(* Logix 5000 project; controller PLC_Safety vendor 1 type 14 code 148 rev 37.11; software revision 37.00; part 2 of 3 *)
(* tags used below, declared in another part *)
   Contador_num_pza : COUNTER;
   Contador_pza_aprove : COUNTER;
   Contador_pza_rechazada : COUNTER;
   Counter_Parts : COUNTER;   // Trazabilidad
   Done_cicle : BOOL;
   FANUC_R1 : BOOL;
   FANUC_R2 : BOOL;
   FANUC_R3 : BOOL;
   FANUC_R4 : BOOL;
   Fanuc_Strobe : BOOL;
   HMI_Cognex_medio : DINT;   // HMI
   HMI_Fanucbrazo : DINT;   // HMI
   HMI_Fanucdelta : DINT;   // HMI
   HMI_Fcognexmedio : BOOL;   // HMI
   HMI_Ffanucbrazo : BOOL;   // HMI
   HMI_Ffanucdelta : BOOL;   // HMI
   HMI_Fplc1 : BOOL;   // HMI
   HMI_Fplc2 : BOOL;   // HMI
   HMI_Fplcseguridad : BOOL;   // HMI
   HMI_kinetix1 : BOOL;   // HMI
   HMI_kinetix2 : BOOL;
   HMI_Kinetix_1 : DINT;   // HMI
   HMI_Kinetix_2 : DINT;
   HMI_PLC1 : DINT;   // HMI
   HMI_PLC2 : DINT;   // HMI
   HMI_PLC_Seguridad : DINT;   // HMI
   HMI_PointIO1 : BOOL;   // HMI
   HMI_PointIO2 : BOOL;
   HMI_PointIO3 : BOOL;
   HMI_PointIO4 : BOOL;
   HMI_PointIO6 : BOOL;
   HMI_PointIO_1 : DINT;   // HMI
   HMI_PointIO_2 : DINT;
   HMI_PointIO_3 : DINT;
   HMI_PointIO_4 : DINT;
   HMI_PointIO_6 : DINT;
   HMI_R_cognex1 : BOOL;
   HMI_R_cognex2 : BOOL;
   HMI_R_PF1 : BOOL;
   HMI_R_PF2 : BOOL;
   HMI_S_cognex1 : BOOL;
   HMI_S_cognex2 : BOOL;
   HMI_S_PF1 : BOOL;
   HMI_S_PF2 : BOOL;
   HMI_Switch1 : BOOL;
   HMI_Switch2 : BOOL;
   HMI_Switch3 : BOOL;
   HMI_Switch4 : BOOL;
   HMI_Switch5 : BOOL;
   OSF_Fault_Reset_Fanuc : BOOL;
   Part : REAL;
   Piece_Approved : BOOL;
   Piece_Base : BOOL;
   Piece_Coil : BOOL;
   Piece_Rejected : BOOL;
   Piece_Upper : BOOL;
   S2_Height_1 : BOOL;
   S2_Height_2 : BOOL;
   S2_Height_3 : BOOL;
   S2_Height_4 : BOOL;
   S2_Height_5 : BOOL;
   S2_Height_6 : BOOL;
   S2_Height_Conveyor_1 : BOOL;
   S2_Height_Conveyor_2 : BOOL;
   S2_MAM_Height_1 : MOTION_INSTRUCTION;
   S2_MAM_Height_2 : MOTION_INSTRUCTION;
   S2_MAM_Height_3 : MOTION_INSTRUCTION;
   S2_MAM_Height_4 : MOTION_INSTRUCTION;
   S2_MAM_Height_5 : MOTION_INSTRUCTION;
   S2_MAM_Height_6 : MOTION_INSTRUCTION;
   S2_MAM_Height_Conveyor_1 : MOTION_INSTRUCTION;
   S2_MAM_Height_Conveyor_2 : MOTION_INSTRUCTION;
   S2_MSO_Storage : MOTION_INSTRUCTION;
   S2_Sensor_Height_1 : BOOL;
   S2_Sensor_Height_2 : BOOL;
   S2_Sensor_Height_3 : BOOL;
   S2_Sensor_Height_4 : BOOL;
   S2_Sensor_Height_5 : BOOL;
   S2_Sensor_Height_6 : BOOL;
   S2_Sensor_Height_Conveyor_1 : BOOL;
   S2_Sensor_Height_Conveyor_2 : BOOL;
   S2_Storage_On : BOOL;
   Sensor_FANUC_R1 : BOOL;
   Sensor_FANUC_R2 : BOOL;
   Sensor_FANUC_R3 : BOOL;
   Sensor_FANUC_R4 : BOOL;
   Start_Button_1_Secuencia : BOOL;
   Start_Button_2_Secuencia : BOOL;
   Start_Button_3_Secuencia : BOOL;
   Trigger_Cognex_3 : BOOL;
   Axis_2 : AXIS_CIP_DRIVE;   // Storage 2
   Data_From_PLC2 : DINT[20];
   Data_To_PLC1 : DINT[20];
   Data_To_PLC2 : DINT[20];
   E_Stop_1_NC : ALIAS FOR Point_IO_Gabinete_1:6:I.Pt01Data;   // E Stop 1 Normally Close
   E_Stop_1_NO : ALIAS FOR Point_IO_Gabinete_1:6:I.Pt00Data;   // E Stop 1 Normally Open
   E_Stop_2_NC : ALIAS FOR Point_IO_Gabinete_2:6:I.Pt01Data;   // E Stop 2 Normally Close
   E_Stop_2_NO : ALIAS FOR Point_IO_Gabinete_2:6:I.Pt00Data;   // E Stop 2 Normally Open
   E_Stop_3_NC : ALIAS FOR Point_IO_Gabinete_6:4:I.Pt02Data;   // E Stop 3 Normally Close
   E_Stop_3_NO : ALIAS FOR Point_IO_Gabinete_6:4:I.Pt03Data;   // E Stop 3 Normally Open
   E_Stop_Conveyor_1_NC : ALIAS FOR Point_IO_Gabinete_3:11:I.Pt00Data;   // E Stop Conveyor 1 Normally Close
   E_Stop_Conveyor_1_NO : ALIAS FOR Point_IO_Gabinete_3:11:I.Pt01Data;   // E Stop Conveyor 1 Normally Open
   E_Stop_Conveyor_2_NC : ALIAS FOR Point_IO_Gabinete_4:11:I.Pt00Data;   // E Stop Conveyor 2 Normally Close
   E_Stop_Conveyor_2_NO : ALIAS FOR Point_IO_Gabinete_4:11:I.Pt01Data;   // E Stop Conveyor 2 Normally Open
   E_Stop_OK : BOOL;
   Reset_General : BOOL;
   Safety_OK : BOOL;
(* MainProgram, continued *)

ROUTINE R05_Storage_2   (* ladder *)
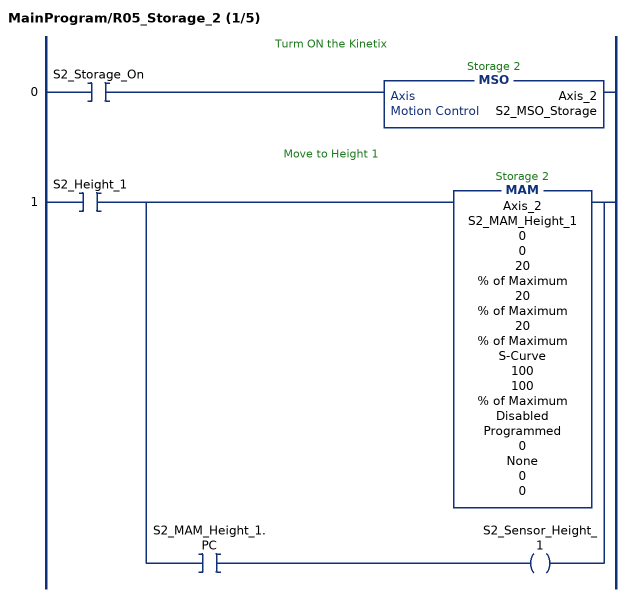
   // Turm ON the Kinetix
   0: XIC(S2_Storage_On)MSO(Axis_2,S2_MSO_Storage);
   // Move to Height 1
   1: XIC(S2_Height_1)[MAM(Axis_2,S2_MAM_Height_1,0,0,20,% of Maximum,20,% of Maximum,20,% of Maximum,S-Curve,100,100,% of Maximum,Disabled,Programmed,0,None,0,0) ,XIC(S2_MAM_Height_1.PC) OTE(S2_Sensor_Height_1) ];
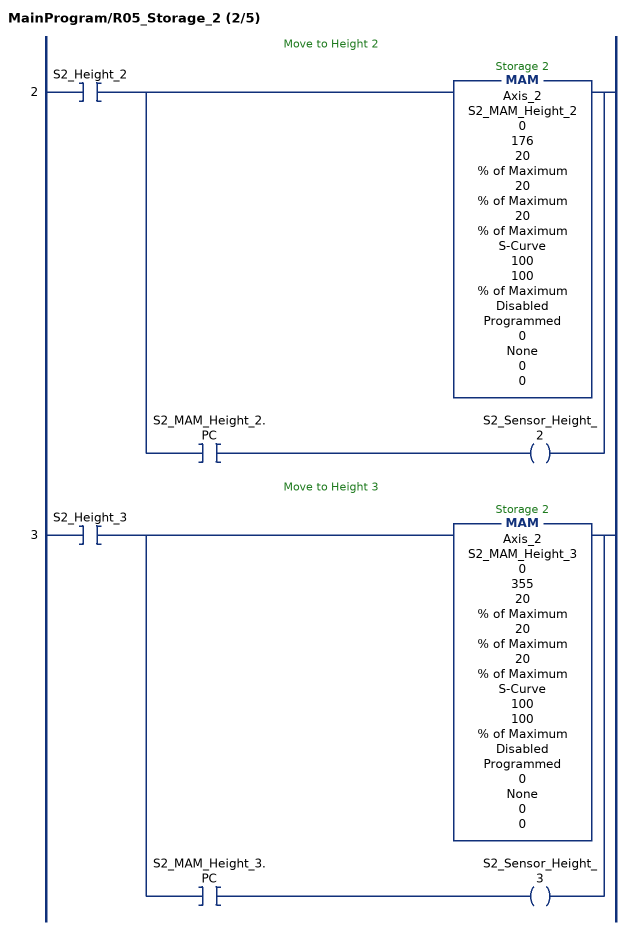
   // Move to Height 2
   2: XIC(S2_Height_2)[MAM(Axis_2,S2_MAM_Height_2,0,176,20,% of Maximum,20,% of Maximum,20,% of Maximum,S-Curve,100,100,% of Maximum,Disabled,Programmed,0,None,0,0) ,XIC(S2_MAM_Height_2.PC) OTE(S2_Sensor_Height_2) ];
   // Move to Height 3
   3: XIC(S2_Height_3)[MAM(Axis_2,S2_MAM_Height_3,0,355,20,% of Maximum,20,% of Maximum,20,% of Maximum,S-Curve,100,100,% of Maximum,Disabled,Programmed,0,None,0,0) ,XIC(S2_MAM_Height_3.PC) OTE(S2_Sensor_Height_3) ];
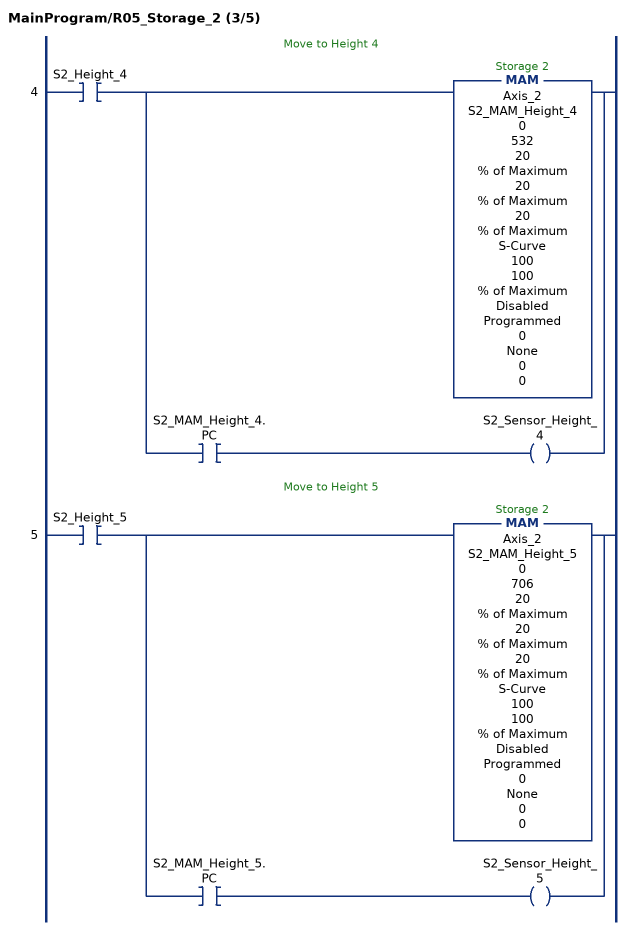
   // Move to Height 4
   4: XIC(S2_Height_4)[MAM(Axis_2,S2_MAM_Height_4,0,532,20,% of Maximum,20,% of Maximum,20,% of Maximum,S-Curve,100,100,% of Maximum,Disabled,Programmed,0,None,0,0) ,XIC(S2_MAM_Height_4.PC) OTE(S2_Sensor_Height_4) ];
   // Move to Height 5
   5: XIC(S2_Height_5)[MAM(Axis_2,S2_MAM_Height_5,0,706,20,% of Maximum,20,% of Maximum,20,% of Maximum,S-Curve,100,100,% of Maximum,Disabled,Programmed,0,None,0,0) ,XIC(S2_MAM_Height_5.PC) OTE(S2_Sensor_Height_5) ];
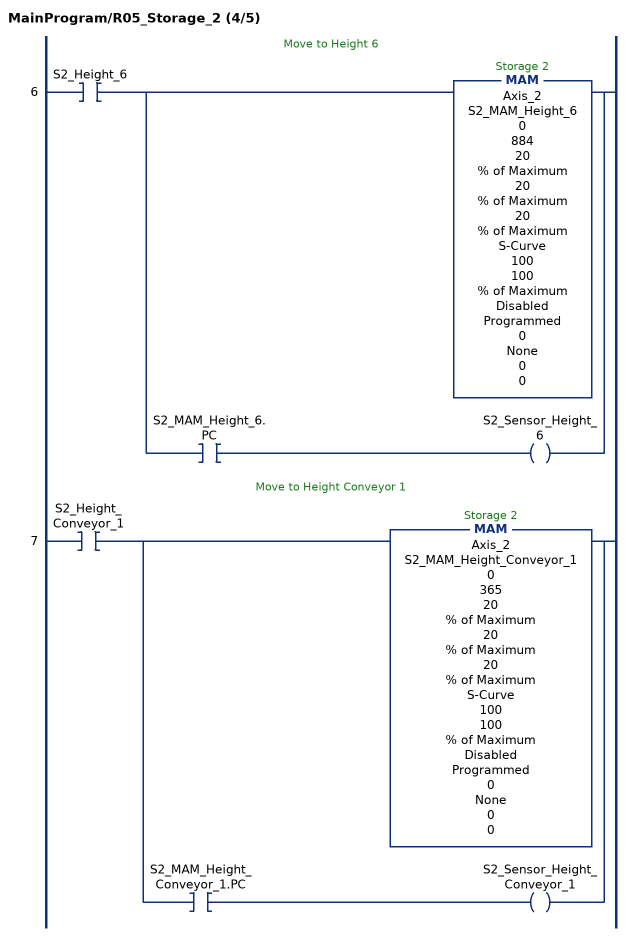
   // Move to Height 6
   6: XIC(S2_Height_6)[MAM(Axis_2,S2_MAM_Height_6,0,884,20,% of Maximum,20,% of Maximum,20,% of Maximum,S-Curve,100,100,% of Maximum,Disabled,Programmed,0,None,0,0) ,XIC(S2_MAM_Height_6.PC) OTE(S2_Sensor_Height_6) ];
   // Move to Height Conveyor 1
   7: XIC(S2_Height_Conveyor_1)[MAM(Axis_2,S2_MAM_Height_Conveyor_1,0,365,20,% of Maximum,20,% of Maximum,20,% of Maximum,S-Curve,100,100,% of Maximum,Disabled,Programmed,0,None,0,0) ,XIC(S2_MAM_Height_Conveyor_1.PC) OTE(S2_Sensor_Height_Conveyor_1) ];
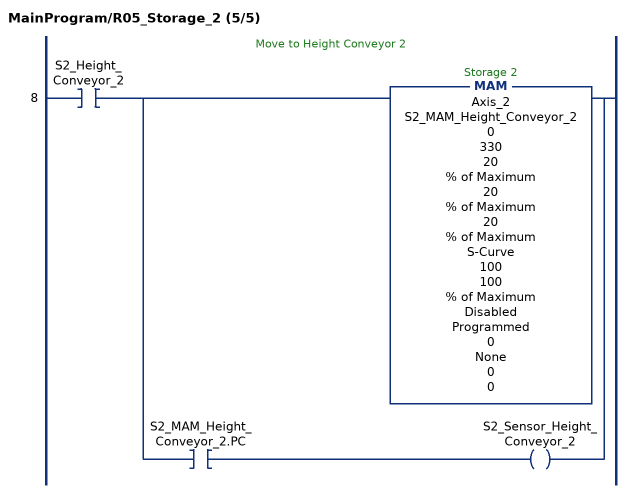
   // Move to Height Conveyor 2
   8: XIC(S2_Height_Conveyor_2)[MAM(Axis_2,S2_MAM_Height_Conveyor_2,0,330,20,% of Maximum,20,% of Maximum,20,% of Maximum,S-Curve,100,100,% of Maximum,Disabled,Programmed,0,None,0,0) ,XIC(S2_MAM_Height_Conveyor_2.PC) OTE(S2_Sensor_Height_Conveyor_2) ];
END_ROUTINE

ROUTINE R06_Fanuc   (* ladder *)
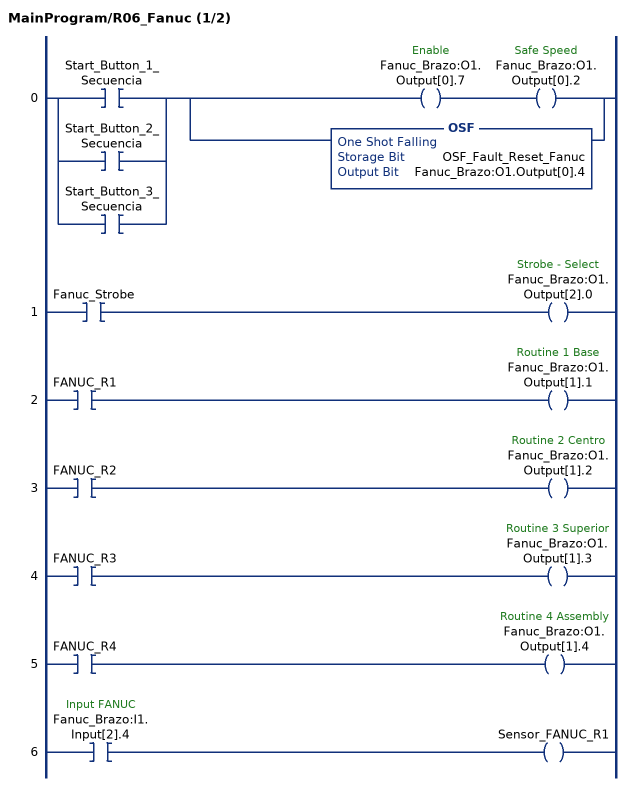
   0: [XIC(Start_Button_1_Secuencia) ,XIC(Start_Button_2_Secuencia) ,XIC(Start_Button_3_Secuencia) ][OTE(Fanuc_Brazo:O1.Output[0].7) OTE(Fanuc_Brazo:O1.Output[0].2) ,OSF(OSF_Fault_Reset_Fanuc,Fanuc_Brazo:O1.Output[0].4) ];
   1: XIC(Fanuc_Strobe)OTE(Fanuc_Brazo:O1.Output[2].0);
   2: XIC(FANUC_R1)OTE(Fanuc_Brazo:O1.Output[1].1);
   3: XIC(FANUC_R2)OTE(Fanuc_Brazo:O1.Output[1].2);
   4: XIC(FANUC_R3)OTE(Fanuc_Brazo:O1.Output[1].3);
   5: XIC(FANUC_R4)OTE(Fanuc_Brazo:O1.Output[1].4);
   6: XIC(Fanuc_Brazo:I1.Input[2].4)OTE(Sensor_FANUC_R1);
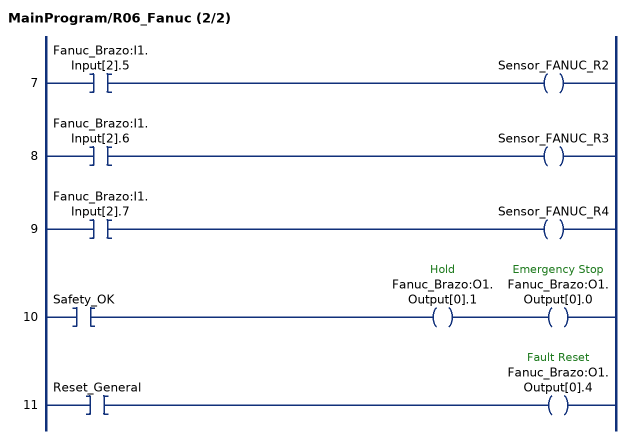
   7: XIC(Fanuc_Brazo:I1.Input[2].5)OTE(Sensor_FANUC_R2);
   8: XIC(Fanuc_Brazo:I1.Input[2].6)OTE(Sensor_FANUC_R3);
   9: XIC(Fanuc_Brazo:I1.Input[2].7)OTE(Sensor_FANUC_R4);
   10: XIC(Safety_OK)OTE(Fanuc_Brazo:O1.Output[0].1)OTE(Fanuc_Brazo:O1.Output[0].0);
   11: XIC(Reset_General)OTE(Fanuc_Brazo:O1.Output[0].4);
END_ROUTINE

ROUTINE R07_Cognex_3   (* ladder *)
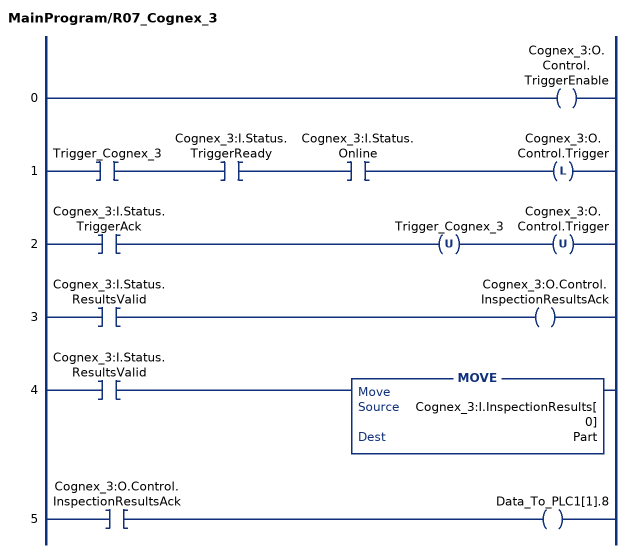
   0: OTE(Cognex_3:O.Control.TriggerEnable);
   1: XIC(Trigger_Cognex_3)XIC(Cognex_3:I.Status.TriggerReady)XIC(Cognex_3:I.Status.Online)OTL(Cognex_3:O.Control.Trigger);
   2: XIC(Cognex_3:I.Status.TriggerAck)OTU(Trigger_Cognex_3)OTU(Cognex_3:O.Control.Trigger);
   3: XIC(Cognex_3:I.Status.ResultsValid)OTE(Cognex_3:O.Control.InspectionResultsAck);
   4: XIC(Cognex_3:I.Status.ResultsValid)MOVE(Cognex_3:I.InspectionResults[0],Part);
   5: XIC(Cognex_3:O.Control.InspectionResultsAck)OTE(Data_To_PLC1[1].8);
END_ROUTINE

ROUTINE R08_Status_Red   (* ladder *)
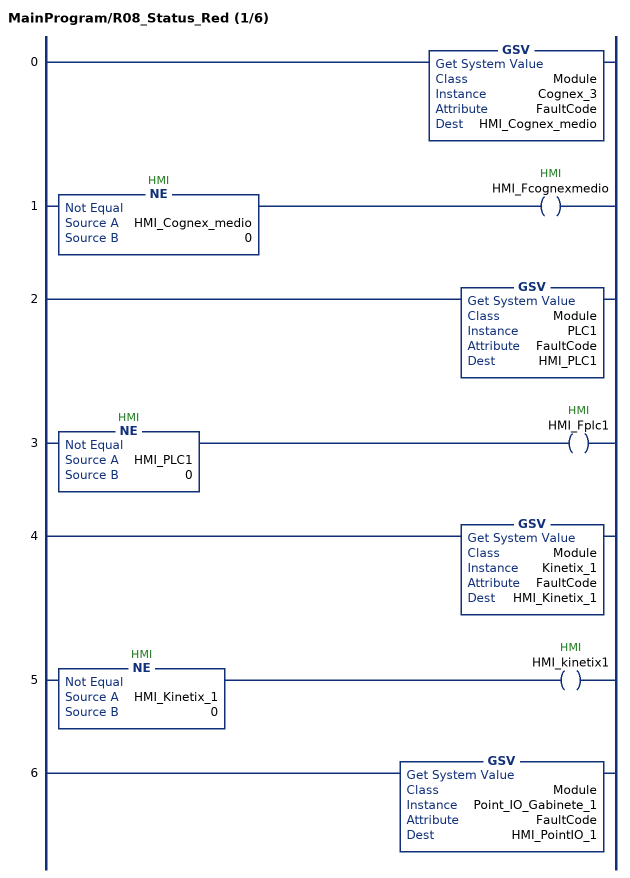
   0: GSV(Module,Cognex_3,FaultCode,HMI_Cognex_medio);
   1: NE(HMI_Cognex_medio,0)OTE(HMI_Fcognexmedio);
   2: GSV(Module,PLC1,FaultCode,HMI_PLC1);
   3: NE(HMI_PLC1,0)OTE(HMI_Fplc1);
   4: GSV(Module,Kinetix_1,FaultCode,HMI_Kinetix_1);
   5: NE(HMI_Kinetix_1,0)OTE(HMI_kinetix1);
   6: GSV(Module,Point_IO_Gabinete_1,FaultCode,HMI_PointIO_1);
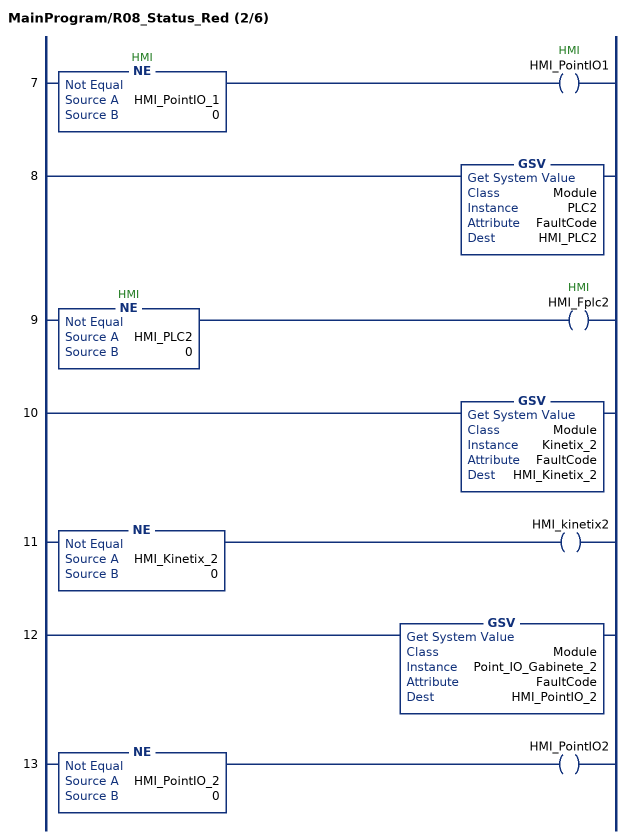
   7: NE(HMI_PointIO_1,0)OTE(HMI_PointIO1);
   8: GSV(Module,PLC2,FaultCode,HMI_PLC2);
   9: NE(HMI_PLC2,0)OTE(HMI_Fplc2);
   10: GSV(Module,Kinetix_2,FaultCode,HMI_Kinetix_2);
   11: NE(HMI_Kinetix_2,0)OTE(HMI_kinetix2);
   12: GSV(Module,Point_IO_Gabinete_2,FaultCode,HMI_PointIO_2);
   13: NE(HMI_PointIO_2,0)OTE(HMI_PointIO2);
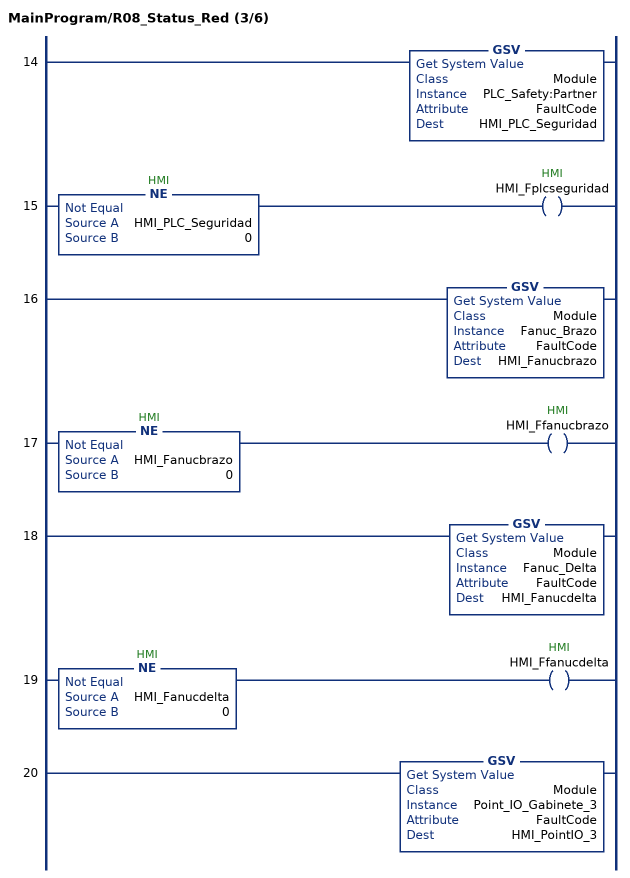
   14: GSV(Module,PLC_Safety:Partner,FaultCode,HMI_PLC_Seguridad);
   15: NE(HMI_PLC_Seguridad,0)OTE(HMI_Fplcseguridad);
   16: GSV(Module,Fanuc_Brazo,FaultCode,HMI_Fanucbrazo);
   17: NE(HMI_Fanucbrazo,0)OTE(HMI_Ffanucbrazo);
   18: GSV(Module,Fanuc_Delta,FaultCode,HMI_Fanucdelta);
   19: NE(HMI_Fanucdelta,0)OTE(HMI_Ffanucdelta);
   20: GSV(Module,Point_IO_Gabinete_3,FaultCode,HMI_PointIO_3);
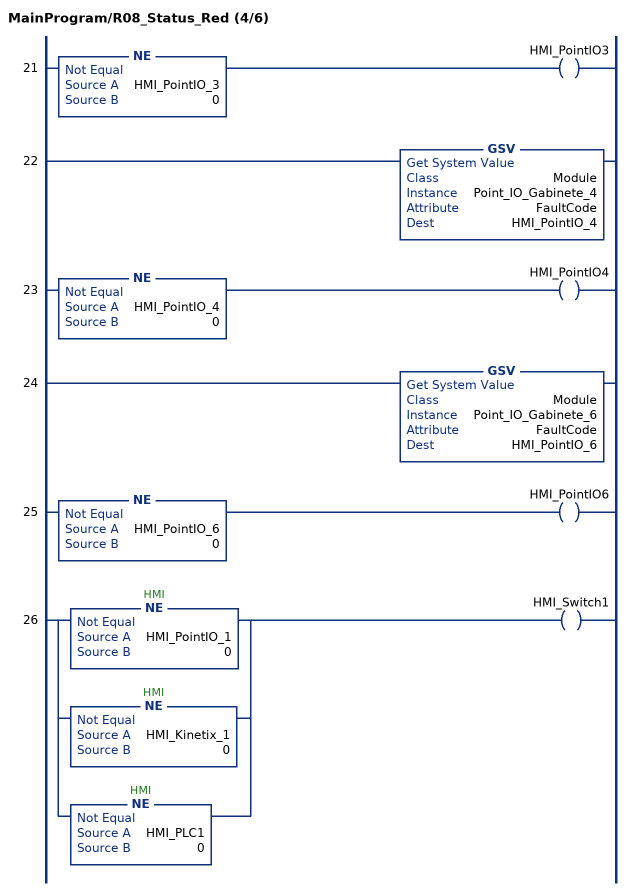
   21: NE(HMI_PointIO_3,0)OTE(HMI_PointIO3);
   22: GSV(Module,Point_IO_Gabinete_4,FaultCode,HMI_PointIO_4);
   23: NE(HMI_PointIO_4,0)OTE(HMI_PointIO4);
   24: GSV(Module,Point_IO_Gabinete_6,FaultCode,HMI_PointIO_6);
   25: NE(HMI_PointIO_6,0)OTE(HMI_PointIO6);
   26: [NE(HMI_PointIO_1,0) ,NE(HMI_Kinetix_1,0) ,NE(HMI_PLC1,0) ]OTE(HMI_Switch1);
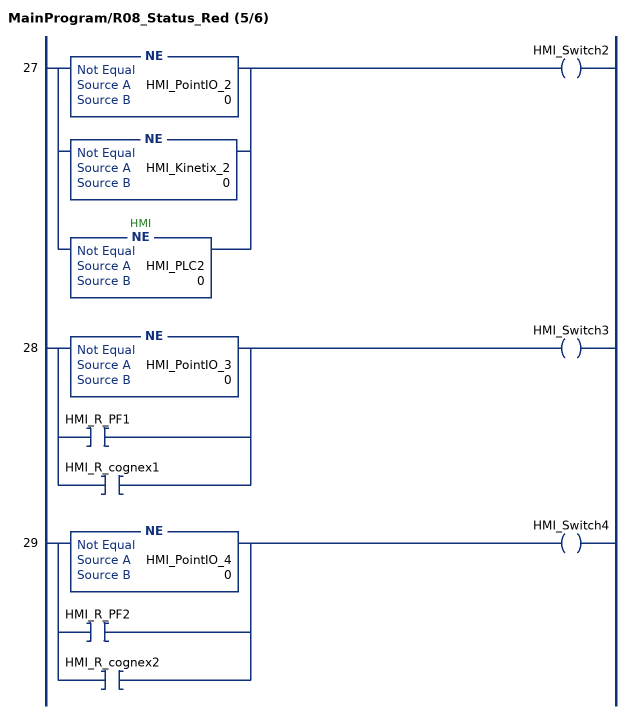
   27: [NE(HMI_PointIO_2,0) ,NE(HMI_Kinetix_2,0) ,NE(HMI_PLC2,0) ]OTE(HMI_Switch2);
   28: [NE(HMI_PointIO_3,0) ,XIC(HMI_R_PF1) ,XIC(HMI_R_cognex1) ]OTE(HMI_Switch3);
   29: [NE(HMI_PointIO_4,0) ,XIC(HMI_R_PF2) ,XIC(HMI_R_cognex2) ]OTE(HMI_Switch4);
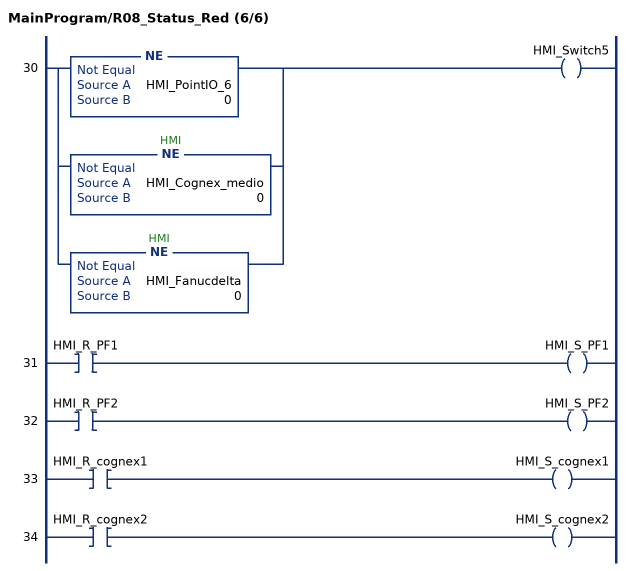
   30: [NE(HMI_PointIO_6,0) ,NE(HMI_Cognex_medio,0) ,NE(HMI_Fanucdelta,0) ]OTE(HMI_Switch5);
   31: XIC(HMI_R_PF1)OTE(HMI_S_PF1);
   32: XIC(HMI_R_PF2)OTE(HMI_S_PF2);
   33: XIC(HMI_R_cognex1)OTE(HMI_S_cognex1);
   34: XIC(HMI_R_cognex2)OTE(HMI_S_cognex2);
END_ROUTINE

ROUTINE R09_Trazabilidad   (* ladder *)
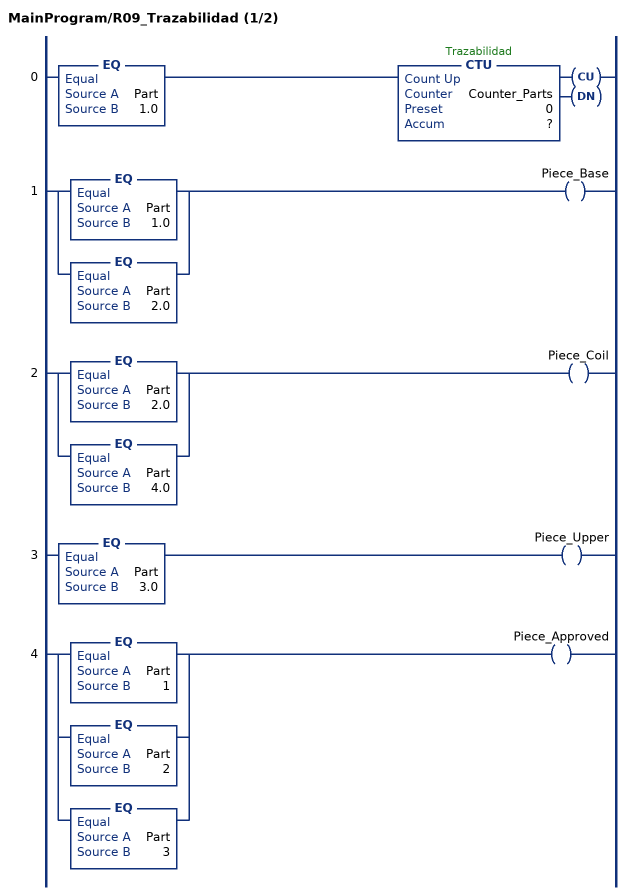
   0: EQ(Part,1.0)CTU(Counter_Parts,?,?);
   1: [EQ(Part,1.0) ,EQ(Part,2.0) ]OTE(Piece_Base);
   2: [EQ(Part,2.0) ,EQ(Part,4.0) ]OTE(Piece_Coil);
   3: EQ(Part,3.0)OTE(Piece_Upper);
   4: [EQ(Part,1) ,EQ(Part,2) ,EQ(Part,3) ]OTE(Piece_Approved);
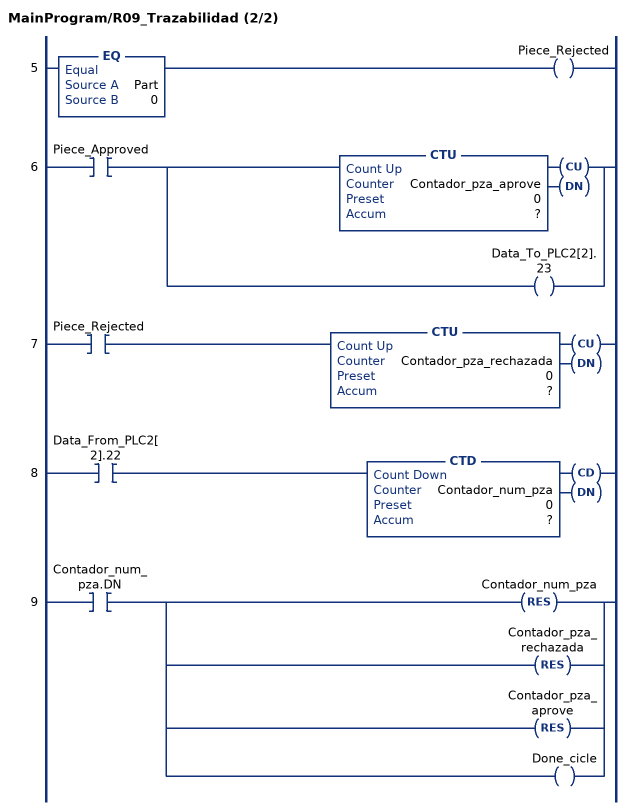
   5: EQ(Part,0)OTE(Piece_Rejected);
   6: XIC(Piece_Approved)[CTU(Contador_pza_aprove,?,?) ,OTE(Data_To_PLC2[2].23) ];
   7: XIC(Piece_Rejected)CTU(Contador_pza_rechazada,?,?);
   8: XIC(Data_From_PLC2[2].22)CTD(Contador_num_pza,?,?);
   9: XIC(Contador_num_pza.DN)[RES(Contador_num_pza) ,RES(Contador_pza_rechazada) ,RES(Contador_pza_aprove) ,OTE(Done_cicle) ];
END_ROUTINE
END_PROGRAM

PROGRAM SafetyProgram   (* main routine R00_Main_Routine, safety *)
VAR
   Auto_OK : BOOL;
   dummy_test : BOOL := 1;
   dummy_test_2 : BOOL := 1;
   dummy_test_3 : BOOL;
   dummy_test_4 : BOOL;
   E_Stop_1 : DCI_STOP := (ChannelA := 1, InputStatus := 1, ColdStartType := 1, InputType := 2, DiscrepancyTime := 500, O1 := 1);
   E_Stop_1_Status_OK : BOOL := 1;
   E_Stop_2 : DCI_STOP := (ChannelA := 1, InputStatus := 1, ColdStartType := 1, InputType := 2, DiscrepancyTime := 500, O1 := 1);
   E_Stop_2_Status_OK : BOOL := 1;
   E_Stop_3 : DCI_STOP := (ChannelA := 1, InputStatus := 1, ColdStartType := 1, InputType := 2, DiscrepancyTime := 150, O1 := 1);
   E_Stop_3_Status_OK : BOOL := 1;
   E_Stop_Conveyor_1 : DCI_STOP := (ChannelA := 1, InputStatus := 1, ColdStartType := 1, InputType := 2, DiscrepancyTime := 150, O1 := 1);
   E_Stop_Conveyor_1_Status_OK : BOOL := 1;
   E_Stop_Conveyor_2 : DCI_STOP := (ChannelA := 1, InputStatus := 1, ColdStartType := 1, InputType := 2, DiscrepancyTime := 150, O1 := 1);
   E_Stop_Conveyor_2_Status_OK : BOOL := 1;
   Fanuc_Enable : BOOL;
   Gate_1 : DCI_STOP := (ChannelA := 1, ChannelB := 1, InputStatus := 1, ColdStartType := 1, SafetyFunction := 1, DiscrepancyTime := 500, O1 := 1);
   Gate_1_State : BOOL := 1;
   Gate_2 : DCI_STOP := (InputStatus := 1, ColdStartType := 1, SafetyFunction := 1, DiscrepancyTime := 500);
   Gate_2_State : BOOL := 1;
   GuardLock_OK : BOOL;
   LightCurtain : DCI_STOP := (ChannelA := 1, ChannelB := 1, InputStatus := 1, ColdStartType := 1, SafetyFunction := 2, DiscrepancyTime := 500, O1 := 1);
   LightCurtain_OK : BOOL := 1;
   LightCurtain_State : BOOL := 1;
   Manual_OK : BOOL := 1;
   OSF_Reset_G1 : BOOL;
   OSF_Reset_G2 : BOOL;
   OSF_Reset_P1 : BOOL;
   OSF_Reset_P2 : BOOL;
   Reset_G1 : BOOL;
   Reset_G2 : BOOL;
   Reset_P1 : BOOL;
   Reset_P2 : BOOL;
   Safety_Mat_OK : BOOL;
   SafetyScanner1 : DCI_STOP := (InputStatus := 1, ColdStartType := 1, SafetyFunction := 3, DiscrepancyTime := 500);
   SafetyScanner1_OK : BOOL;
   SafetyScanner1_State : BOOL := 1;
   SafetyScanner2 : DCI_STOP := (InputStatus := 1, ColdStartType := 1, SafetyFunction := 3, DiscrepancyTime := 500);
   SafetyScanner2_OK : BOOL;
   SafetyScanner2_State : BOOL := 1;
   Servo_Drive_1_Enable : BOOL;
   Servo_Drive_1_Safety : CONFIGURABLE_ROUT := (Actuate := 1, FeedbackType := 1, InputStatus := 1, OutputStatus := 1, FeedbackReactionTime := 500, FP := 1, FaultCode := 32);
   Servo_Drive_1_Status_OK : BOOL := 1;
   Servo_Drive_2_Enable : BOOL;
   Servo_Drive_2_Safety : CONFIGURABLE_ROUT := (Actuate := 1, FeedbackType := 1, InputStatus := 1, OutputStatus := 1, FeedbackReactionTime := 500, FP := 1, FaultCode := 32);
   Servo_Drive_2_Status_OK : BOOL := 1;
   true : BOOL := 1;
   VFD_1_Enable : BOOL;
   VFD_1_Safety : CONFIGURABLE_ROUT := (Actuate := 1, FeedbackType := 1, InputStatus := 1, OutputStatus := 1, FeedbackReactionTime := 500, FP := 1, FaultCode := 32);
   VFD_1_Status_OK : BOOL := 1;
   VFD_2_Enable : BOOL;
   VFD_2_Safety : CONFIGURABLE_ROUT := (Actuate := 1, FeedbackType := 1, InputStatus := 1, OutputStatus := 1, FeedbackReactionTime := 500, FP := 1, FaultCode := 32);
   VFD_2_Status_OK : BOOL := 1;
END_VAR

ROUTINE R00_Main_Routine   (* ladder *)
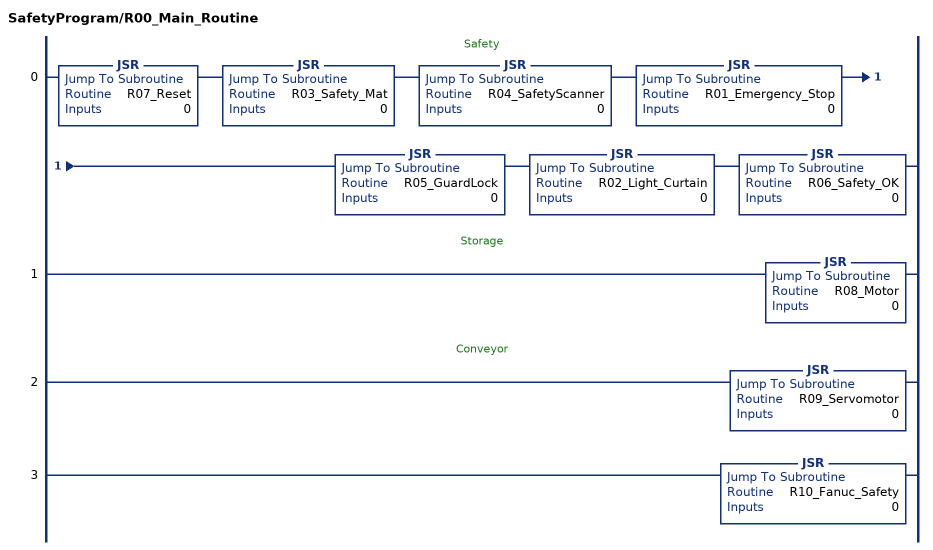
   // Safety
   0: JSR(R07_Reset,0)JSR(R03_Safety_Mat,0)JSR(R04_SafetyScanner,0)JSR(R01_Emergency_Stop,0)JSR(R05_GuardLock,0)JSR(R02_Light_Curtain,0)JSR(R06_Safety_OK,0);
   // Storage
   1: JSR(R08_Motor,0);
   // Conveyor
   2: JSR(R09_Servomotor,0);
   3: JSR(R10_Fanuc_Safety,0);
END_ROUTINE

ROUTINE R01_Emergency_Stop   (* ladder *)
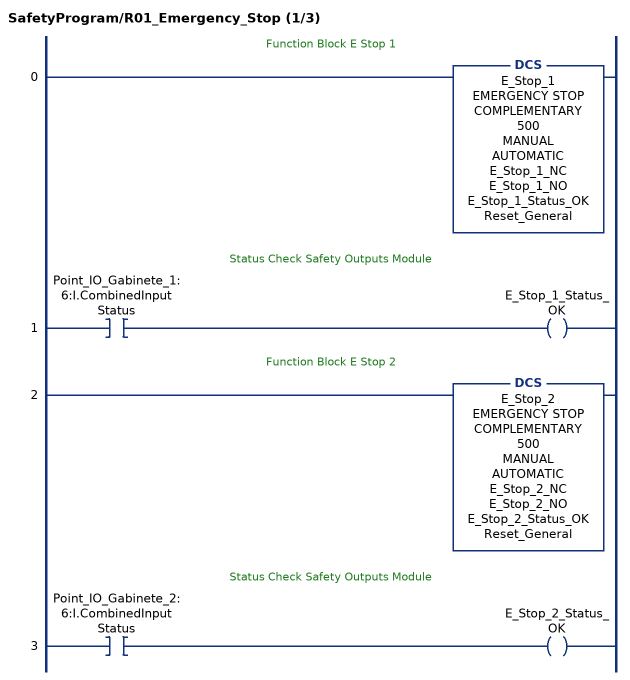
   // Function Block E Stop 1
   0: DCS(E_Stop_1,EMERGENCY STOP,COMPLEMENTARY,500,MANUAL,AUTOMATIC,E_Stop_1_NC,E_Stop_1_NO,E_Stop_1_Status_OK,Reset_General);
   // Status Check Safety Outputs Module
   1: XIC(Point_IO_Gabinete_1:6:I.CombinedInputStatus)OTE(E_Stop_1_Status_OK);
   // Function Block E Stop 2
   2: DCS(E_Stop_2,EMERGENCY STOP,COMPLEMENTARY,500,MANUAL,AUTOMATIC,E_Stop_2_NC,E_Stop_2_NO,E_Stop_2_Status_OK,Reset_General);
   // Status Check Safety Outputs Module
   3: XIC(Point_IO_Gabinete_2:6:I.CombinedInputStatus)OTE(E_Stop_2_Status_OK);
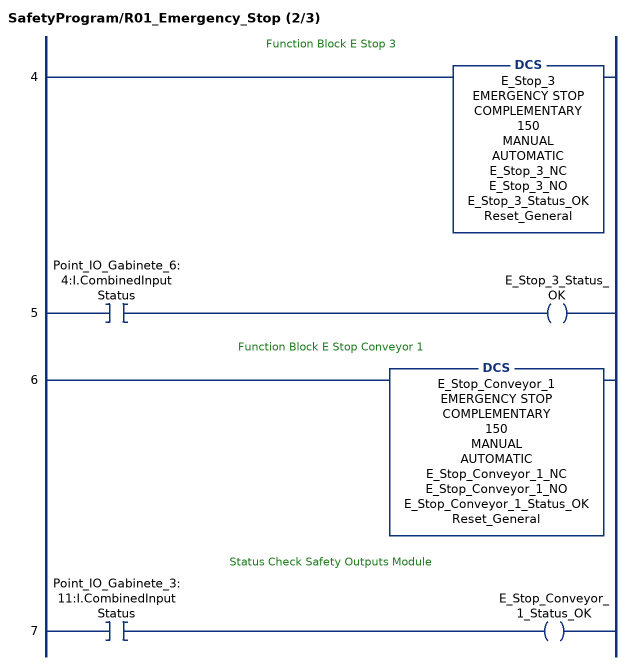
   // Function Block E Stop 3
   4: DCS(E_Stop_3,EMERGENCY STOP,COMPLEMENTARY,150,MANUAL,AUTOMATIC,E_Stop_3_NC,E_Stop_3_NO,E_Stop_3_Status_OK,Reset_General);
   5: XIC(Point_IO_Gabinete_6:4:I.CombinedInputStatus)OTE(E_Stop_3_Status_OK);
   // Function Block E Stop Conveyor 1
   6: DCS(E_Stop_Conveyor_1,EMERGENCY STOP,COMPLEMENTARY,150,MANUAL,AUTOMATIC,E_Stop_Conveyor_1_NC,E_Stop_Conveyor_1_NO,E_Stop_Conveyor_1_Status_OK,Reset_General);
   // Status Check Safety Outputs Module
   7: XIC(Point_IO_Gabinete_3:11:I.CombinedInputStatus)OTE(E_Stop_Conveyor_1_Status_OK);
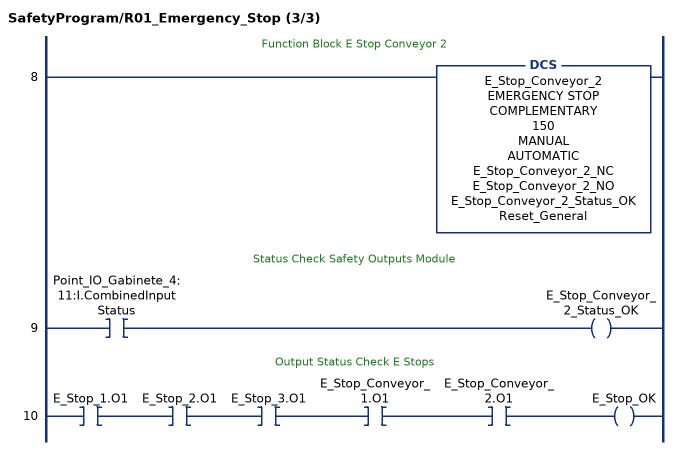
   // Function Block E Stop Conveyor 2
   8: DCS(E_Stop_Conveyor_2,EMERGENCY STOP,COMPLEMENTARY,150,MANUAL,AUTOMATIC,E_Stop_Conveyor_2_NC,E_Stop_Conveyor_2_NO,E_Stop_Conveyor_2_Status_OK,Reset_General);
   // Status Check Safety Outputs Module
   9: XIC(Point_IO_Gabinete_4:11:I.CombinedInputStatus)OTE(E_Stop_Conveyor_2_Status_OK);
   // Output Status Check E Stops
   10: XIC(E_Stop_1.O1)XIC(E_Stop_2.O1)XIC(E_Stop_3.O1)XIC(E_Stop_Conveyor_1.O1)XIC(E_Stop_Conveyor_2.O1)OTE(E_Stop_OK);
END_ROUTINE
